{attribute 'no_check'}
//°/s -> RPM
FUNCTION DEGREES_TO_RPM : LREAL
VAR_INPUT
	IN														:	LREAL;	//Input value
END_VAR
VAR
END_VAR

DEGREES_TO_RPM 											:= IN * 60.0 / 360.0;

END_FUNCTION

(* stored: Version 1.1.0.1, ProductVersion 3.1.4020.12
   POU DEGREES_TO_RPM: Id {b7be0bc0-9381-49e0-b960-9d46fcd9a08f}, SpecialFunc None *)
